TYPE ST_SettingMachinePart01 :
STRUCT
    nMotorType : BYTE; //Motor type
    stMotorSettings : ST_StandardMotorSettings;
    nCylinderType : BYTE; //Cylinder type
    stCylinderSettings : ST_StandardCylinderSettings;
END_STRUCT
END_TYPE

(* stored: Version 1.1.0.1, ProductVersion 3.1.4019.2
   DUT ST_SettingMachinePart01: Id {2b743166-5ec9-4cbc-8481-fd18b58b43db} *)
